// TwinCAT 3 PLC project OEF_5
// ProgramVersion: 3.1.4024.0
// libraries:
//   Tc2_Standard, * (Beckhoff Automation GmbH)
//   Tc2_System, * (Beckhoff Automation GmbH)
//   Tc3_Module, * (Beckhoff Automation GmbH)
// project tree:
//   / PlcTask.TcTTO
//   POUs/ MAIN.TcPOU
// (motion and I/O tree: see PLC project oef_1)
// real-time tasks:
//   TASK PlcTask: cycle T#10ms, priority 20, ADS port 350
//   TASK PlcTask1: cycle T#10ms, priority 21, ADS port 351
//   TASK PlcTask2: cycle T#10ms, priority 22, ADS port 352
//   TASK PlcTask3: cycle T#10ms, priority 23, ADS port 353
//   TASK PlcTask4: cycle T#10ms, priority 24, ADS port 354
//   TASK PlcTask5: cycle T#10ms, priority 25, ADS port 355
//   TASK PlcTask6: cycle T#10ms, priority 26, ADS port 356
// variable links:
//   OEF_5/OEF_5 Instance <-> Device 1 (EtherCAT)/Term 1 (EK1200)/Term 3 (EL2008)
//     PlcTask Outputs/MAIN.bLED1 <-> Channel 2/Output

CONFIGURATION OEF_5
    RESOURCE PLC ON TwinCAT3
        TASK PlcTask(INTERVAL := T#10ms, PRIORITY := 25);
        PROGRAM MAIN WITH PlcTask : MAIN;
    END_RESOURCE
END_CONFIGURATION

// ---- POUs/MAIN.TcPOU
PROGRAM MAIN
VAR
	fbTP1: TP := (PT := TIME#500MS);
	fbTP2: TP := (PT := TIME#500MS);
	bLED1 AT %Q*: BOOL := false;
END_VAR

fbTP1(IN:= not(fbTP2.Q), Q=> bLED1);
fbTP2(IN:= not(fbTP1.Q));

END_PROGRAM
